Fanuc TP program (LS listing): PNS0001.LS

/PROG  PNS0001
/ATTR
OWNER		= MNEDITOR;
COMMENT		= "";
PROG_SIZE	= 179;
CREATE		= DATE 18-04-05  TIME 09:30:08;
MODIFIED	= DATE 18-04-05  TIME 09:53:42;
FILE_NAME	= ;
VERSION		= 0;
LINE_COUNT	= 1;
MEMORY_SIZE	= 555;
PROTECT		= READ;
TCD:  STACK_SIZE	= 0,
      TASK_PRIORITY	= 50,
      TIME_SLICE	= 0,
      BUSY_LAMP_OFF	= 0,
      ABORT_REQUEST	= 0,
      PAUSE_REQUEST	= 0;
DEFAULT_GROUP	= 1,*,*,*,*;
CONTROL_CODE	= 00000000 00000000;
/APPL

AUTO_SINGULARITY_HEADER;
  ENABLE_SINGULARITY_AVOIDANCE   : FALSE;
/MN
   1:  CALL MAIN    ;
/POS
/END
